{attribute 'qualified_only'}
VAR_GLOBAL CONSTANT
	Unknown		: T_PackMLMode := 0;
	Manual		: T_PackMLMode := 1;
	Production	: T_PackMLMode := 2;
END_VAR

(* stored: Version 1.1.0.1, ProductVersion 3.1.4026.18
   GVL GVL_PackMLMode: Id {2a3de17e-afb4-4382-91ef-cd097cfb9a0e} *)
